{attribute 'linkalways'} 
{attribute 'no_explicit_call' := 'This FB is a CLASS and must be accessed using methods or properties'}
{attribute 'enable_dynamic_creation'}
FUNCTION_BLOCK LinkedListNode EXTENDS Disposable IMPLEMENTS I_LinkedListNode
VAR
	pBuffer : POINTER TO BYTE;
	bufferSize : UDINT;
	_previous : I_LinkedListNode;
	_next : I_LinkedListNode;
END_VAR

METHOD PRIVATE CopyBufferToDestination
VAR_INPUT
	DestinationAddress : PVOID;
END_VAR
MEMCPY(DestinationAddress, pBuffer, bufferSize);
END_METHOD

METHOD PRIVATE CopySourceToBuffer
VAR_INPUT
	SourceAddress : PVOID;
END_VAR
MEMCPY(pBuffer, SourceAddress, bufferSize);
END_METHOD

METHOD PRIVATE CreateBuffer
VAR_INPUT
	SizeInBytes : UDINT;
END_VAR
bufferSize := SizeInBytes;
pBuffer := __NEW(BYTE, SizeInBytes);
END_METHOD

PROPERTY PUBLIC DataSize : UDINT
GET // PUBLIC
DataSize := bufferSize;
END_GET
END_PROPERTY

METHOD PRIVATE DestroyBuffer
IF pBuffer = 0 THEN
	RETURN;
END_IF

__DELETE(pBuffer);
bufferSize := 0;
END_METHOD

METHOD PUBLIC Equals : BOOL
VAR_INPUT
	Symbol : ANY;
END_VAR
IF pBuffer = 0 THEN
	RETURN;
END_IF

IF bufferSize <> DINT_TO_UDINT(Symbol.diSize) THEN
	RETURN;
END_IF

Equals := MEMCMP(Symbol.pValue, pBuffer, bufferSize) = 0;
END_METHOD

METHOD FB_exit : BOOL
VAR_INPUT
	bInCopyCode : BOOL; // if TRUE, the exit method is called for exiting an instance that is copied afterwards (online change).
END_VAR
IF bInCopyCode THEN
	RETURN;
END_IF

DestroyBuffer();
END_METHOD

METHOD FB_init : BOOL
VAR_INPUT
	bInitRetains : BOOL; // if TRUE, the retain variables are initialized (warm start / cold start)
	bInCopyCode : BOOL;  // if TRUE, the instance afterwards gets moved into the copy code (online change)
	Source : ANY;
END_VAR
CreateBuffer(DINT_TO_UDINT(Source.diSize));
CopySourceToBuffer(Source.pValue);
END_METHOD

PROPERTY PUBLIC Next : I_LinkedListNode
GET // PUBLIC
Next := _next;
END_GET
SET // PUBLIC
_next := Next;
END_SET
END_PROPERTY

PROPERTY PUBLIC Previous : I_LinkedListNode
GET // PUBLIC
Previous := _previous;
END_GET
SET // PUBLIC
_previous := Previous;
END_SET
END_PROPERTY

METHOD PUBLIC TryGet : BOOL;
VAR_INPUT
	Destination : ANY;
END_VAR
TryGet := TryGetTo(Destination.pValue, DINT_TO_UDINT(Destination.diSize));
END_METHOD

METHOD PUBLIC TryGetTo : BOOL;
VAR_INPUT
	DestinationAddress : PVOID;
	DestinationSize : UDINT;
END_VAR
IF pBuffer = 0 THEN
	RETURN;
END_IF

IF bufferSize <> DestinationSize THEN
	RETURN;
END_IF

CopyBufferToDestination(DestinationAddress);
TryGetTo := TRUE;
END_METHOD

END_FUNCTION_BLOCK

(* stored: Version 1.1.0.1, ProductVersion 3.1.4024.12
   POU LinkedListNode: Id {a22f637d-88c7-419b-b580-90cbbca9b84f}, SpecialFunc None
   Folder Constructor: Id {20b6c8a5-1664-49d8-b5bd-9c1711ef40ca}
   Folder Destructor: Id {11cc8ede-e096-43a1-8b10-0aa5baa00abd}
   Folder Private: Id {22c2c466-04ff-4ebc-8087-51bcece35ac8}
   Method CopyBufferToDestination: Id {fa8fa4ca-2673-4587-b20a-5d8baba6e8e2}
   Method CopySourceToBuffer: Id {18cfb4cb-e3f8-45eb-a9a7-ca95cb406a85}
   Method CreateBuffer: Id {7d892977-21cd-4a4e-a73c-403e3b2efbf2}
   Property DataSize: Id {32500e6c-c7d3-4d2c-84c1-5f4f96b638ab}
   Get Get: Id {4192d556-9198-433f-8448-000b91c96e74}
   Method DestroyBuffer: Id {c7c49d2f-9f6d-45dd-bd4d-86f1f8ec2952}
   Method Equals: Id {3dae5d6f-b48a-45e9-9190-dda6a3aca1f0}
   Method FB_exit: Id {8bebc509-1cf0-4449-be85-11d2862d71e7}
   Method FB_init: Id {773c76da-ef84-49fb-b4c4-dad69385c1c1}
   Property Next: Id {8b27ac43-47ee-4572-8701-fb684f77d844}
   Get Get: Id {05c22ed3-2d83-4489-89cf-363f8dd84840}
   Set Set: Id {a0b2ce1d-a978-4ac1-849f-de98ceb46fb9}
   Property Previous: Id {e0c608ca-4ce5-46c6-9f68-957bb0262213}
   Get Get: Id {5bc37a05-92b7-4f4f-b921-88dbf94828f9}
   Set Set: Id {afd8fd71-1240-4ef0-9b3a-7bb0d9e593a6}
   Method TryGet: Id {2e237f93-18af-4ede-ae4f-657387db0b35}
   Method TryGetTo: Id {fc1682a2-75fe-45fb-bb00-791b41822df9} *)
